RoboDK station: Drone_simulator.rdk

Station Drone_simulator (saved by RoboDK 5.4.0). Poses are relative to the parent item; angles as X-Y-Z fixed-axis rotations.
